// TIA Portal project "S7_elevador_3pisos v2" (V14)

(* hardware
DEVICE "S7-1200 station_1"  S7-1200 Station
   slot 0: "Rack_0"  Rack  V1.0
   slot 1: "PLC_1"  CPU 1212C AC/DC/Rly  6ES7 212-1BE40-0XB0  V4.2
*)

// ===== PLC "PLC_1"  CPU 1212C AC/DC/Rly =====

VAR_GLOBAL   // PLC tag table "Default tag table"
   "Sinalização P1" AT %Q0.3 : Bool;
   "Sensor RC" AT %I0.3 : Bool;
   "Sinalização RC" AT %Q0.2 : Bool;
   "Sensor P1" AT %I0.4 : Bool;
   "Sensor P2" AT %I0.5 : Bool;
   "Sinalização P2" AT %Q0.4 : Bool;
   "Saída Livre" AT %Q0.5 : Bool;
   "Início" AT %M0.1 : Bool;
   "Seleção Piso" AT %M0.2 : Bool;
   "Entrada Livre" AT %I0.7 : Bool;
   "Porta Aberta" AT %I0.6 : Bool;
   "Motor DOWN" AT %Q0.1 : Bool;
   "Posição RC" AT %M1.0 : Bool;
   "Posição P1" AT %M1.1 : Bool;
   "Posição P2" AT %M1.2 : Bool;
   "Botão RC" AT %I0.0 : Bool;
   "Botão P1" AT %I0.1 : Bool;
   "Botão P2" AT %I0.2 : Bool;
   "Move RC" AT %M2.0 : Bool;
   "Move P1" AT %M2.1 : Bool;
   "Move P2" AT %M2.2 : Bool;
   "Subir" AT %M2.3 : Bool;
   "Descer" AT %M2.4 : Bool;
   "Motor UP" AT %Q0.0 : Bool;
END_VAR

ORGANIZATION_BLOCK "Main"   // OB1, LAD, ProgramCycle
TITLE = "Main Program Sweep (Cycle)"
{ S7_Optimized_Access := 'TRUE' }
VERSION : 0.1
   VAR_INPUT
      Initial_Call : Bool;   // Initial call of this OB
      Remanence : Bool;   // =True, if remanent data are available
   END_VAR
BEGIN

REGION Network 1: Início
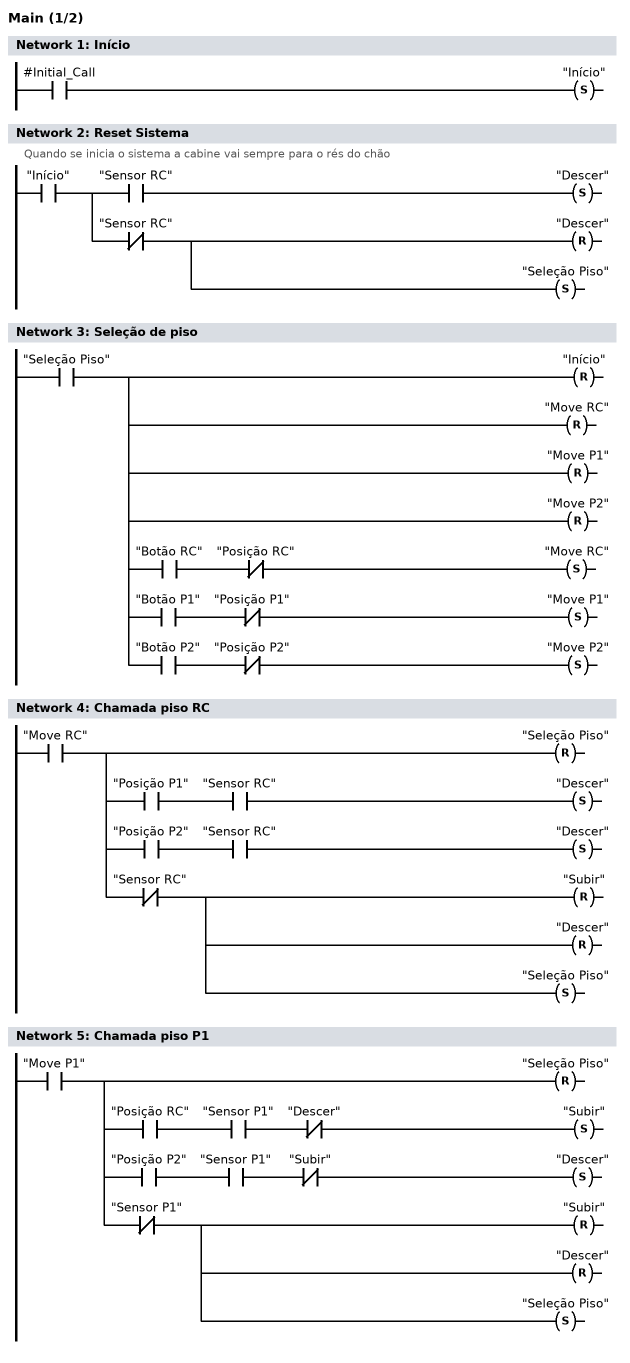
   RUNG wire#powerrail
      Contact( #Initial_Call )
      S_Coil( "Início" )
   END_RUNG
   // the same network as SCL:
   IF #Initial_Call THEN "Início" := TRUE; END_IF;
END_REGION

REGION Network 2: Reset Sistema
   // Quando se inicia o sistema a cabine vai sempre para o rés do chão
   RUNG wire#powerrail
      Contact( "Início" )
      wire#w1
      Contact( "Sensor RC" )
      S_Coil( "Descer" )
   END_RUNG
   RUNG wire#w1
      I_Contact( "Sensor RC" )
      wire#w2
      R_Coil( "Descer" )
   END_RUNG
   RUNG wire#w2
      S_Coil( "Seleção Piso" )
   END_RUNG
   // the same network as SCL:
   IF "Início" AND "Sensor RC" THEN "Descer" := TRUE; END_IF;
   IF "Início" AND NOT "Sensor RC" THEN
       "Descer" := FALSE;
       "Seleção Piso" := TRUE;
   END_IF;
END_REGION

REGION Network 3: Seleção de piso
   RUNG wire#powerrail
      Contact( "Seleção Piso" )
      wire#w1
      R_Coil( "Início" )
   END_RUNG
   RUNG wire#w1
      R_Coil( "Move RC" )
   END_RUNG
   RUNG wire#w1
      R_Coil( "Move P1" )
   END_RUNG
   RUNG wire#w1
      R_Coil( "Move P2" )
   END_RUNG
   RUNG wire#w1
      Contact( "Botão RC" )
      I_Contact( "Posição RC" )
      S_Coil( "Move RC" )
   END_RUNG
   RUNG wire#w1
      Contact( "Botão P1" )
      I_Contact( "Posição P1" )
      S_Coil( "Move P1" )
   END_RUNG
   RUNG wire#w1
      Contact( "Botão P2" )
      I_Contact( "Posição P2" )
      S_Coil( "Move P2" )
   END_RUNG
   // the same network as SCL:
   IF "Seleção Piso" THEN
       "Início" := FALSE;
       "Move RC" := FALSE;
       "Move P1" := FALSE;
       "Move P2" := FALSE;
   END_IF;
   IF "Seleção Piso" AND "Botão RC" AND NOT "Posição RC" THEN "Move RC" := TRUE; END_IF;
   IF "Seleção Piso" AND "Botão P1" AND NOT "Posição P1" THEN "Move P1" := TRUE; END_IF;
   IF "Seleção Piso" AND "Botão P2" AND NOT "Posição P2" THEN "Move P2" := TRUE; END_IF;
END_REGION

REGION Network 4: Chamada piso RC
   RUNG wire#powerrail
      Contact( "Move RC" )
      wire#w1
      R_Coil( "Seleção Piso" )
   END_RUNG
   RUNG wire#w1
      Contact( "Posição P1" )
      Contact( "Sensor RC" )
      S_Coil( "Descer" )
   END_RUNG
   RUNG wire#w1
      Contact( "Posição P2" )
      Contact( "Sensor RC" )
      S_Coil( "Descer" )
   END_RUNG
   RUNG wire#w1
      I_Contact( "Sensor RC" )
      wire#w2
      R_Coil( "Subir" )
   END_RUNG
   RUNG wire#w2
      R_Coil( "Descer" )
   END_RUNG
   RUNG wire#w2
      S_Coil( "Seleção Piso" )
   END_RUNG
   // the same network as SCL:
   IF "Move RC" THEN "Seleção Piso" := FALSE; END_IF;
   IF "Move RC" AND "Posição P1" AND "Sensor RC" THEN "Descer" := TRUE; END_IF;
   IF "Move RC" AND "Posição P2" AND "Sensor RC" THEN "Descer" := TRUE; END_IF;
   IF "Move RC" AND NOT "Sensor RC" THEN
       "Subir" := FALSE;
       "Descer" := FALSE;
       "Seleção Piso" := TRUE;
   END_IF;
END_REGION

REGION Network 5: Chamada piso P1
   RUNG wire#powerrail
      Contact( "Move P1" )
      wire#w1
      R_Coil( "Seleção Piso" )
   END_RUNG
   RUNG wire#w1
      Contact( "Posição RC" )
      Contact( "Sensor P1" )
      I_Contact( "Descer" )
      S_Coil( "Subir" )
   END_RUNG
   RUNG wire#w1
      Contact( "Posição P2" )
      Contact( "Sensor P1" )
      I_Contact( "Subir" )
      S_Coil( "Descer" )
   END_RUNG
   RUNG wire#w1
      I_Contact( "Sensor P1" )
      wire#w2
      R_Coil( "Subir" )
   END_RUNG
   RUNG wire#w2
      R_Coil( "Descer" )
   END_RUNG
   RUNG wire#w2
      S_Coil( "Seleção Piso" )
   END_RUNG
   // the same network as SCL:
   IF "Move P1" THEN "Seleção Piso" := FALSE; END_IF;
   IF "Move P1" AND "Posição RC" AND "Sensor P1" AND NOT "Descer" THEN "Subir" := TRUE; END_IF;
   IF "Move P1" AND "Posição P2" AND "Sensor P1" AND NOT "Subir" THEN "Descer" := TRUE; END_IF;
   IF "Move P1" AND NOT "Sensor P1" THEN
       "Subir" := FALSE;
       "Descer" := FALSE;
       "Seleção Piso" := TRUE;
   END_IF;
END_REGION

REGION Network 6: Chamada piso P2
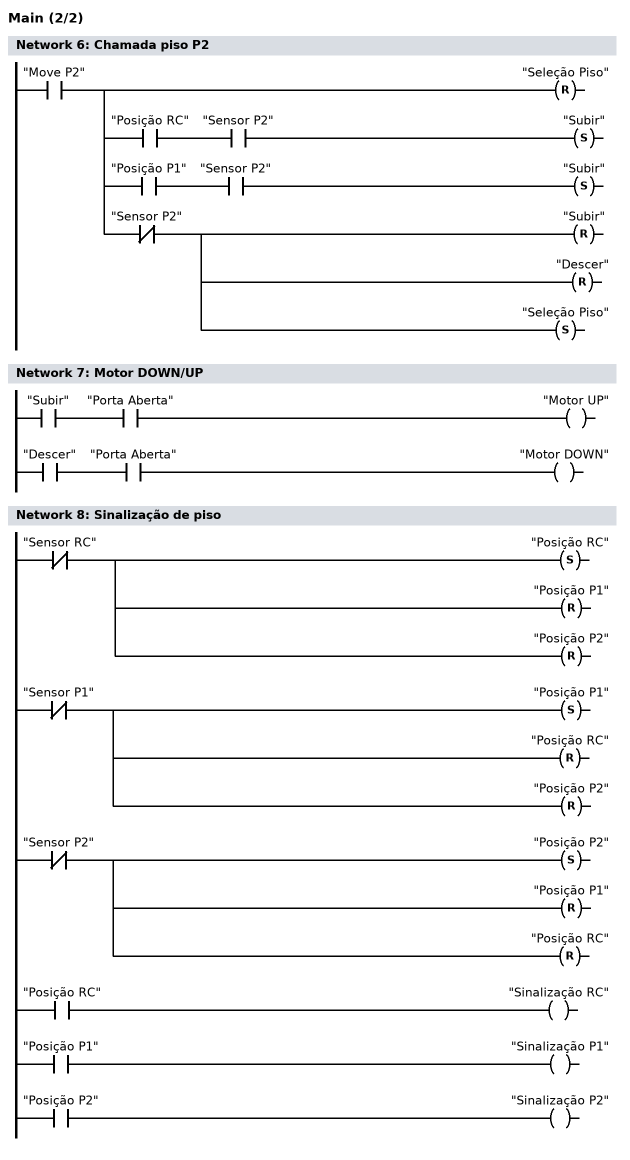
   RUNG wire#powerrail
      Contact( "Move P2" )
      wire#w1
      R_Coil( "Seleção Piso" )
   END_RUNG
   RUNG wire#w1
      Contact( "Posição RC" )
      Contact( "Sensor P2" )
      S_Coil( "Subir" )
   END_RUNG
   RUNG wire#w1
      Contact( "Posição P1" )
      Contact( "Sensor P2" )
      S_Coil( "Subir" )
   END_RUNG
   RUNG wire#w1
      I_Contact( "Sensor P2" )
      wire#w2
      R_Coil( "Subir" )
   END_RUNG
   RUNG wire#w2
      R_Coil( "Descer" )
   END_RUNG
   RUNG wire#w2
      S_Coil( "Seleção Piso" )
   END_RUNG
   // the same network as SCL:
   IF "Move P2" THEN "Seleção Piso" := FALSE; END_IF;
   IF "Move P2" AND "Posição RC" AND "Sensor P2" THEN "Subir" := TRUE; END_IF;
   IF "Move P2" AND "Posição P1" AND "Sensor P2" THEN "Subir" := TRUE; END_IF;
   IF "Move P2" AND NOT "Sensor P2" THEN
       "Subir" := FALSE;
       "Descer" := FALSE;
       "Seleção Piso" := TRUE;
   END_IF;
END_REGION

REGION Network 7: Motor DOWN/UP
   RUNG wire#powerrail
      Contact( "Subir" )
      Contact( "Porta Aberta" )
      Coil( "Motor UP" )
   END_RUNG
   RUNG wire#powerrail
      Contact( "Descer" )
      Contact( "Porta Aberta" )
      Coil( "Motor DOWN" )
   END_RUNG
   // the same network as SCL:
   "Motor UP" := "Subir" AND "Porta Aberta";
   "Motor DOWN" := "Descer" AND "Porta Aberta";
END_REGION

REGION Network 8: Sinalização de piso
   RUNG wire#powerrail
      I_Contact( "Sensor RC" )
      wire#w1
      S_Coil( "Posição RC" )
   END_RUNG
   RUNG wire#w1
      R_Coil( "Posição P1" )
   END_RUNG
   RUNG wire#w1
      R_Coil( "Posição P2" )
   END_RUNG
   RUNG wire#powerrail
      I_Contact( "Sensor P1" )
      wire#w2
      S_Coil( "Posição P1" )
   END_RUNG
   RUNG wire#w2
      R_Coil( "Posição RC" )
   END_RUNG
   RUNG wire#w2
      R_Coil( "Posição P2" )
   END_RUNG
   RUNG wire#powerrail
      I_Contact( "Sensor P2" )
      wire#w3
      S_Coil( "Posição P2" )
   END_RUNG
   RUNG wire#w3
      R_Coil( "Posição P1" )
   END_RUNG
   RUNG wire#w3
      R_Coil( "Posição RC" )
   END_RUNG
   RUNG wire#powerrail
      Contact( "Posição RC" )
      Coil( "Sinalização RC" )
   END_RUNG
   RUNG wire#powerrail
      Contact( "Posição P1" )
      Coil( "Sinalização P1" )
   END_RUNG
   RUNG wire#powerrail
      Contact( "Posição P2" )
      Coil( "Sinalização P2" )
   END_RUNG
   // the same network as SCL:
   IF NOT "Sensor RC" THEN
       "Posição RC" := TRUE;
       "Posição P1" := FALSE;
       "Posição P2" := FALSE;
   END_IF;
   IF NOT "Sensor P1" THEN
       "Posição P1" := TRUE;
       "Posição RC" := FALSE;
       "Posição P2" := FALSE;
   END_IF;
   IF NOT "Sensor P2" THEN
       "Posição P2" := TRUE;
       "Posição P1" := FALSE;
       "Posição RC" := FALSE;
   END_IF;
   "Sinalização RC" := "Posição RC";
   "Sinalização P1" := "Posição P1";
   "Sinalização P2" := "Posição P2";
END_REGION
END_ORGANIZATION_BLOCK